(* CODESYS project 2019-01-16 Thingsboard Demo V04.ecp

Project tree, tasks and I/O mapping:
  PFC200 : 750-8202 PFC200 2ETH RS, WAGO, order no. 0750-8202, version 5.13.2.22
    application Application
      libraries: ; CIP Encapsulation Layer, * (3S - Smart Software Solutions GmbH); WagoAppJSON, 1.0.1.1 (WAGO); WagoSysLog, 1.0.1.0 (WAGO); WagoAppCloud, 1.3.0.7 (WAGO)
      task PLC_Task (cyclic, interval t#50ms, priority 15) calls PLC_PRG
      task VISU_TASK (cyclic, interval 100 ms, priority 15) calls VisuElems.Visu_Prg
      program PLC_PRG [ST]
      image pool ImagePool
      function block showFillingLevel [ST]
      visualisation Visualization
      01_Cloud/
        program NativeMQTT_Publish [ST]
        program JSON_Converter [ST]
    Kbus : Kbus, WAGO, version 1.4.0.2
        unmapped channels: K-BUS diagnostics
    MODBUS
      MODBUS : MODBUS, WAGO, order no. n/a, version 1.1.1.15
    Serial
      COM1 : COM1, WAGO, version 0.0.0.19
  PFC200_G2 : 750-8212 PFC200 2ETH RS, WAGO, order no. 0750-8212, version 5.13.2.22
    application Application
      libraries: ; WagoAppCloud, * (WAGO); WagoAppJSON, 1.0.1.1 (WAGO)
      task PLC_Task (cyclic, interval t#50ms, priority 15) calls PLC_PRG
      program PLC_PRG [FBD]
      program PRG_Build_JSON [ST]
      program PRG_NativeMQTT [ST]
    Common.PCI
    Kbus : Kbus, WAGO, version 1.4.0.2
        unmapped channels: K-BUS diagnostics
      _16_DI_Generic : 075x-16DI, WAGO, order no. 075x-16DI, version 0.0.0.13
          settings: K-BUS Module slot index = 1
          unmapped channels: _IN
      _16_DO_Generic : 075x-16DO, WAGO, order no. 075x-16DO, version 0.0.0.13
          settings: K-BUS Module slot index = 2
          unmapped channels: _OUT
      _4AO_4_20mA : 0750-0555, WAGO, order no. 0750-0555, version 0.0.0.12
          settings: K-BUS Module slot index = 3
          unmapped channels: _QW 1, _QW 2, _QW 3, _QW 4
      _2AI_TC_K_Diagn_Adjust : 0750-0469/0003-0000, WAGO, order no. 0750-0469/0003-0000, version 0.0.0.9
          settings: K-BUS Module slot index = 4
          input  iRawThermo_1 : INT  // _IINT 1
          input  iRawThermo_2 : INT  // _IINT 2
      _2AI_0_10_VDC_SE : 0750-0467, WAGO, order no. 0750-0467, version 0.0.0.9
          settings: K-BUS Module slot index = 5
          input  wRohVoltage_1 : WORD  // _IW 1
          unmapped channels: _IW 2
      _2AO_0_10_VDC : 0750-0550, WAGO, order no. 0750-0550, version 0.0.0.9
          settings: K-BUS Module slot index = 6
          unmapped channels: _QW 1, _QW 2
    MODBUS
      MODBUS : MODBUS, WAGO, order no. n/a, version 1.1.1.15
    Serial
      COM1 : COM1, WAGO, version 0.0.0.19
  libraries: VisuSymbols, 3.5.10.0 (System); WagoVisuIcons, 1.0.1.0 (WAGO)
  text list GlobalTextList
  5ce3da45-db07-42e7-a21c-a00fff4ed8f6|Bilder\Lupe.PNG
  5ce3da45-db07-42e7-a21c-a00fff4ed8f6|Bilder\WAGO_2017_SPS_Messe_Saftfabrik_Freigestellt.png
  5ce3da45-db07-42e7-a21c-a00fff4ed8f6|Bilder\Tank_00_0398.png
  5ce3da45-db07-42e7-a21c-a00fff4ed8f6|Bilder\Tank_10_0398.png
  5ce3da45-db07-42e7-a21c-a00fff4ed8f6|Bilder\Tank_20_0398.png
  5ce3da45-db07-42e7-a21c-a00fff4ed8f6|Bilder\Tank_30_0398.png
  5ce3da45-db07-42e7-a21c-a00fff4ed8f6|Bilder\Tank_40_0398.png
  5ce3da45-db07-42e7-a21c-a00fff4ed8f6|Bilder\Tank_50_0398.png
  5ce3da45-db07-42e7-a21c-a00fff4ed8f6|Bilder\Tank_60_0398.png
  5ce3da45-db07-42e7-a21c-a00fff4ed8f6|Bilder\Tank_70_0398.png
  5ce3da45-db07-42e7-a21c-a00fff4ed8f6|Bilder\Tank_80_0398.png
  5ce3da45-db07-42e7-a21c-a00fff4ed8f6|Bilder\Tank_90_0398.png
  5ce3da45-db07-42e7-a21c-a00fff4ed8f6|Bilder\Tank_100_0398.png
*)

// PFC200/Application/PLC_PRG
PROGRAM PLC_PRG

VAR
	tank1:showFillingLevel;
	sollLevelTank1:INT:=0;
	imageTank1:STRING:='';

	tank2:showFillingLevel;
	sollLevelTank2:INT:=0;
	imageTank2:STRING:='';

	tank3:showFillingLevel;
	sollLevelTank3:INT:=0;
	imageTank3:STRING:='';
	
END_VAR

VAR CONSTANT

END_VAR



tank1(sollLevel:=sollLevelTank1);
imageTank1:=tank1.actualImage;

tank2(sollLevel:=sollLevelTank2);
imageTank2:=tank2.actualImage;

tank3(sollLevel:=sollLevelTank3);
imageTank3:=tank3.actualImage;

NativeMQTT_Publish(levelTank1:=sollLevelTank1,levelTank2:=sollLevelTank2,levelTank3:=sollLevelTank3);

END_PROGRAM

// PFC200/Application/01_Cloud/NativeMQTT_Publish
PROGRAM NativeMQTT_Publish
VAR_INPUT
	levelTank1:INT:=0;
	levelTank2:INT:=0;
	levelTank3:INT:=0;	
END_VAR

VAR
	MyPublishInterval	: TIME := T#5S;
	Timer				: TON;
	
	dwMyCounter 	: DWORD := 1;
	MyString 		: STRING(255);
	MyString1 		: STRING(255);
	aBuffer			: ARRAY[0..255] OF BYTE;
	dwBytesCount 	: DWORD;
	
	oFbPublish 		: WagoAppCloud.FbPublishMQTT;
	xMyTrigger		: BOOL := FALSE;
	dwTimerCounter	: DWORD := 0;
	dwBusyCounter	: DWORD := 0;
	dwErrorCounter	: DWORD := 0;
	
	oldLevel1:INT:=0;
	oldLevel2:INT:=0;
	oldLevel3:INT:=0;
	trigger:BOOL:=FALSE;
	
	//STATUS INFORMATION
	oFbStatus 			: WagoAppCloud.FbStatus_NativeMQTT;
	xMyError			: BOOL := FALSE;
	xConnectedToMyCloud	: BOOL := FALSE;
	rMyFillLevel		: REAL := 0;
	uliMyOutgoingBlocks	: ULINT := 0;

	//JSONLIB
	fbjson: WagoAppJSON.Fb_JSON_Writer_01;
END_VAR

IF ((oldLevel1 = levelTank1) AND (oldLevel2 = levelTank2) AND (oldLevel3 = levelTank3)) THEN
	trigger:=FALSE; 
ELSE
	trigger:=TRUE;
END_IF

Timer(IN := TRUE, PT := MyPublishInterval);
IF (Timer.Q AND trigger) THEN
	Timer(IN := FALSE);
	dwTimerCounter := dwTimerCounter + 1;

	xMyTrigger := trigger;
	oldLevel1:=levelTank1;
	oldLevel2:=levelTank2;
	oldLevel3:=levelTank3;
	IF NOT oFbPublish.xBusy THEN
(*
//JSON Payload via String-Funktionen erstellen
		MyString := '{"LevelTank1": ';
		MyString := CONCAT(MyString, INT_TO_STRING(levelTank1));
		MyString := CONCAT(MyString, ', ');
		
		MyString := CONCAT(MyString, '"LevelTank2": ');
		MyString := CONCAT(MyString, INT_TO_STRING(levelTank2));
		MyString := CONCAT(MyString, ', ');
		
		MyString := CONCAT(MyString, '"LevelTank3": ');
		MyString := CONCAT(MyString, INT_TO_STRING(levelTank3));
		MyString := CONCAT(MyString, '}');
*)

// Alternative: JSON Payload via JSON Lib erstellen
		JSON_Converter(levelTank1:=levelTank1, levelTank2:=levelTank2, levelTank3:=levelTank3, trigger:=trigger);
		MyString := JSON_Converter.sOutput;

		dwBytesCount := Length(MyString);
		MemCopy(pDest := ADR(aBuffer), pSource := ADR(MyString), udiSize := dwBytesCount);
	ELSE
		dwBusyCounter := dwBusyCounter + 1;
	END_IF
	
	IF oFbPublish.xError THEN
		dwErrorCounter := dwErrorCounter + 1;
	END_IF
	
END_IF

oFbPublish(sTopic := 'v1/devices/me/telemetry',
			eQualityOfService := 1,
			dwSize := dwBytesCount,
			aData := aBuffer,
			xTrigger := xMyTrigger);
			
// STATUS INFORMATION	
oFbStatus(xEnabled := TRUE,
		   xError => xMyError,
		   xCloudConnected => xConnectedToMyCloud,			// Will be FALSE after network timeout occured 
		   rCacheFillLevel => rMyFillLevel,					// Increasing value indicates bad network or overload
		   uliOutgoingDataBlocks => uliMyOutgoingBlocks);  	// Only for QoS 1 and 2. Increasing value indicates bad network or overload

// Depending on your internet connection quality, broker performance et. the publish interval will be set here
CASE uliMyOutgoingBlocks OF
	0..10:
		MyPublishInterval := T#50MS;
	11..20:
		MyPublishInterval := T#100MS;
	21..50:
		MyPublishInterval := T#200MS;
	51..100:
		MyPublishInterval := T#500MS;
	101..200:
		MyPublishInterval := T#1000MS;
	201..300:
		MyPublishInterval := T#5000MS;
END_CASE

END_PROGRAM

// PFC200/Application/01_Cloud/JSON_Converter
PROGRAM JSON_Converter
VAR_INPUT
	levelTank1:INT:=0;
	levelTank2:INT:=0;
	levelTank3:INT:=0;	
	trigger:BOOL:=TRUE;
END_VAR
VAR
	fbjson: WagoAppJSON.Fb_JSON_Writer_01;
	MyTemplateString :STRING(1000) := '{"LevelTank1": "#Parameter","LevelTank2": "#Parameter","LevelTank3": "#Parameter"}';
	MyValueArray: ARRAY [0..2] OF STRING;
	xTrig: BOOL := TRUE;
	sOutput: STRING(JSON_MAX_STRING);
END_VAR

MyValueArray[0]:=INT_TO_STRING(levelTank1);
MyValueArray[1]:=INT_TO_STRING(levelTank2);
MyValueArray[2]:=INT_TO_STRING(levelTank3);

fbjson(
	sJSON_BaseFrame:= MyTemplateString,
	oStatus=> , 
	xError=> , 
	xDone=> , 
	aParameterValues:= MyValueArray, 
	xTrigger:= trigger, 
	sOutput:= sOutput);

END_PROGRAM

// PFC200_G2/Application/PLC_PRG
PROGRAM PLC_PRG
VAR
END_VAR

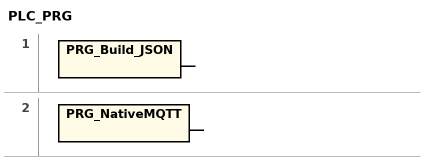
// NETWORK 1
PRG_Build_JSON();

// NETWORK 2
PRG_NativeMQTT();

END_PROGRAM

// PFC200_G2/Application/PRG_Build_JSON
PROGRAM PRG_Build_JSON
VAR
	oFb_JSON: WagoAppJSON.Fb_JSON_Writer_01;
	MyTemplateString :STRING(1000) := 
					'{"Temperature": "#Parameter","Voltage": "#Parameter","Counting Number": "#Parameter"}';
					// "#Parameter" will be replaced with the array value starting by array index"0" to "2"			
	asMyValueArray	: ARRAY [0..2] OF STRING;
	sOutput			: STRING(JSON_MAX_STRING);
	bMyValue		: BYTE := 1;
END_VAR

VAR_INPUT
	xTrigger_Update_Payload: BOOL := TRUE;
END_VAR

//Values for "#Parameter"
asMyValueArray[0]:= TO_STRING(15000/10.0);
asMyValueArray[1]:= TO_STRING(5000*2.3/327.6);
asMyValueArray[2]:= TO_STRING(bMyValue);
bMyValue:=bMyValue+1;


oFb_JSON(
	sJSON_BaseFrame:=MyTemplateString , 
	aParameterValues:= asMyValueArray, 
	xTrigger:= xTrigger_Update_Payload, 
	sOutput:=sOutput );

END_PROGRAM

// PFC200_G2/Application/PRG_NativeMQTT
PROGRAM PRG_NativeMQTT
VAR
	oFbPublishNativeMQTT	: WagoAppCloud.FbPublishMQTT;
	oFbStatusNativeMQTT		: WagoAppCloud.FbStatus_NativeMQTT;
	MyString				: STRING(JSON_MAX_STRING);
	dwBytesCount			: UDINT;
	abBuffer				: ARRAY[0..255] OF BYTE;
	xTrigger_Publish		: BOOL := TRUE;
	xBusy_Publish			: BOOL;
	xError_Publish			: BOOL;
	oStatus_Publish			: FbResult;
	xError_Status_MQTT		: BOOL;
	xCloudConnected			: BOOL;
	rCacheFillLevel			: REAL;
	uliOutgoingDataBlocks	: ULINT;
	oTON: Standard.TON;
END_VAR

oTON(IN:=NOT oTON.Q , PT:= T#1S);
IF oTON.Q THEN
	xTrigger_Publish:=TRUE;
	PRG_Build_JSON.xTrigger_Update_Payload:=TRUE;
END_IF

MyString := PRG_Build_JSON.sOutput;
dwBytesCount := Length(MyString);
MemCopy(pDest := ADR(abBuffer), pSource := ADR(MyString), udiSize := dwBytesCount);

oFbPublishNativeMQTT(
	sTopic:='v1/devices/me/telemetry' ,  //--> https://thingsboard.io/docs/reference/mqtt-api/
	eQualityOfService:= eQualityOfService.QoS1, 
	xRetain:= , 
	dwSize:= dwBytesCount, 
	aData:= abBuffer, 
	xTrigger:= xTrigger_Publish, 
	xBusy=> xBusy_Publish , 
	xError=> xError_Publish, 
	oStatus=> oStatus_Publish);

oFbStatusNativeMQTT(
	xEnabled:= TRUE, 
	xError=> xError_Status_MQTT, 
	xCloudConnected=> xCloudConnected, 
	rCacheFillLevel=> rCacheFillLevel, 
	uliOutgoingDataBlocks=> uliOutgoingDataBlocks);

END_PROGRAM

// PFC200/Application/showFillingLevel
FUNCTION_BLOCK showFillingLevel
VAR_INPUT
	sollLevel:INT:=0;
END_VAR

VAR_OUTPUT
	actualImage:STRING:='Tank1_01';
END_VAR

VAR
	istLevel:INT:=0;
END_VAR

VAR CONSTANT
END_VAR

	CASE sollLevel OF
		0:
			actualImage:='Tank1_00';
		1:
			actualImage:='Tank1_01';
		2:
			actualImage:='Tank1_02';
		3:
			actualImage:='Tank1_03';
		4:
			actualImage:='Tank1_04';
		5:
			actualImage:='Tank1_05';
		6:
			actualImage:='Tank1_06';
		7:
			actualImage:='Tank1_07';
		8:
			actualImage:='Tank1_08';
		9:
			actualImage:='Tank1_09';
		10:
			actualImage:='Tank1_10';			
	END_CASE

END_FUNCTION_BLOCK

// PFC200/Application/Visualization
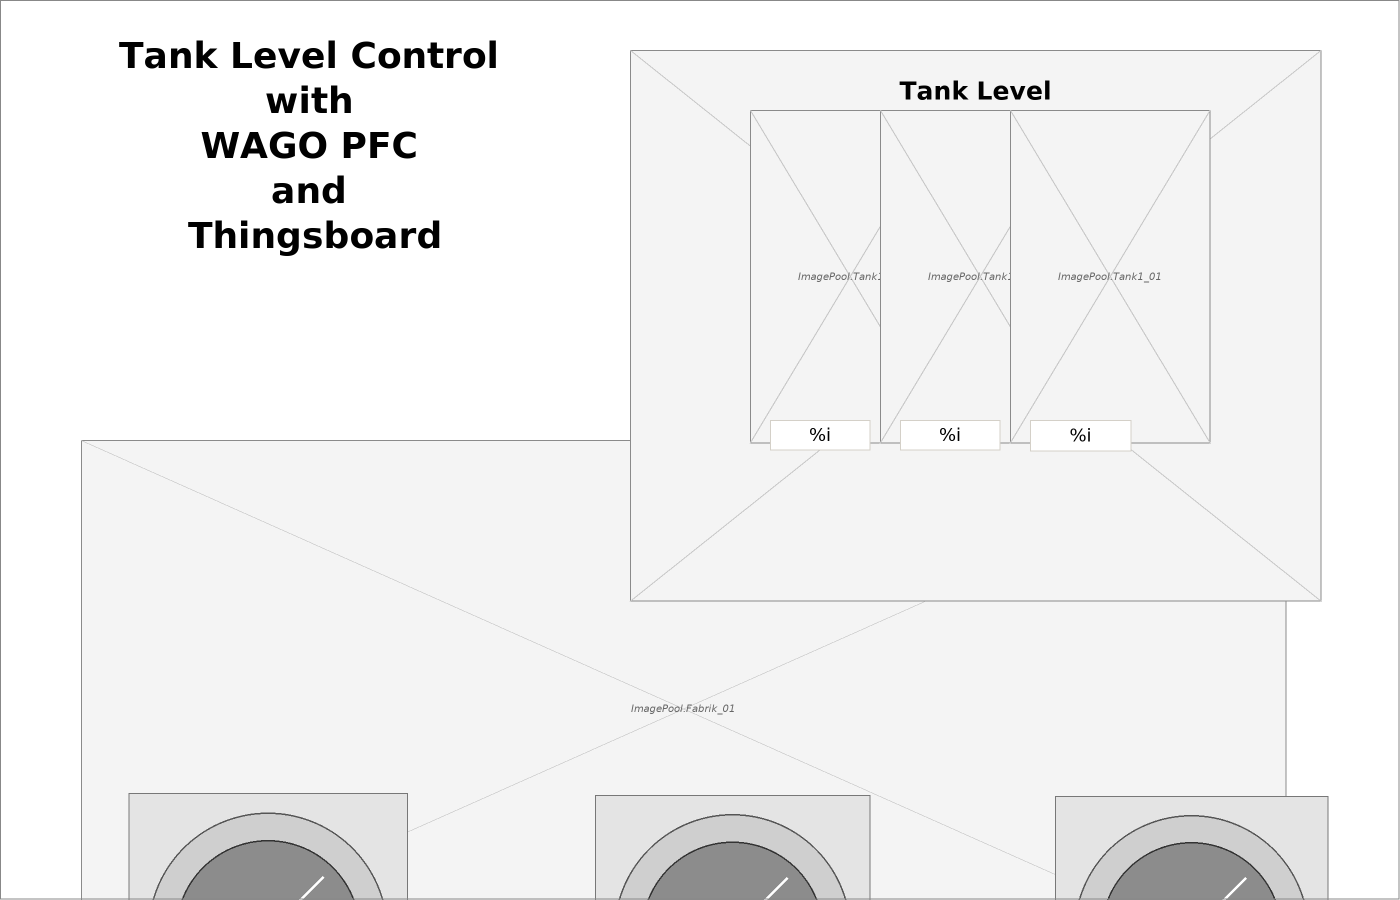
VISUALIZATION Visualization  // 1400x900
    Image (81,440 1205x537), image: ImagePool.Fabrik_01
    Image (630,50 691x551), image: ImagePool.Lupe
    Image (750,110 200x333), image: ImagePool.Tank1_01
        p84334746: PLC_PRG.imageTank1
    Image (880,110 200x333), image: ImagePool.Tank1_01
        p84334746: PLC_PRG.imageTank2
    Image (1010,110 200x333), image: ImagePool.Tank1_01
        p84334746: PLC_PRG.imageTank3
    Label (40,10 551x271), "Tank Level Control with WAGO PFC and Thingsboard"
    Textfield (770,420 100x30), "%i", text variable: PLC_PRG.sollLevelTank1
    Label (890,80 171x21), "Tank Level"
    Textfield (900,420 100x30), "%i", text variable: PLC_PRG.sollLevelTank2
    Textfield (1030,420 101x31), "%i", text variable: PLC_PRG.sollLevelTank3
    Potentiometer360 (122,793 292x279), variable: PLC_PRG.sollLevelTank1, style: Potentiometer-Potentiometer360-Gray, scale format: %.1f, scale 0..10
        p2431819421: Outside
    Potentiometer360 (568,795 329x275), variable: PLC_PRG.sollLevelTank2, style: Potentiometer-Potentiometer360-Gray, scale format: %.1f, scale 0..10
        p2431819421: Outside
    Potentiometer360 (1051,796 281x273), variable: PLC_PRG.sollLevelTank3, style: Potentiometer-Potentiometer360-Gray, scale format: %.1f, scale 0..10
        p2431819421: Outside
END_VISUALIZATION
